(* IEC 61131-3 sources: PortalRobot/Portal_robot/Device/application/FB (part 4) *)

(* ---- FB_MAGAZINE.UpdateTypeStatus.st ---- *)
METHOD PRIVATE UpdateTypeStatus
VAR_IN_OUT
	stMagazineInventory : ST_MAGAZINE_INVENTORY;
END_VAR
VAR
	uiType : UINT; // Тип секции, 1..3
	uiSlot : UINT; // Проверяемый слот
	iSlot  : SINT; // Индекс массива содержимого
END_VAR

// --- BEGIN IMPLEMENTATION ---

FOR uiType := UINT#1 TO UINT#3 DO
	Status.stTypeStatus.aiBlankSlot[uiType] := SINT#0;
	Status.stTypeStatus.aiFreeSlot[uiType] := SINT#0;
	Status.stTypeStatus.auiBlankCount[uiType] := UINT#0;
	Status.stTypeStatus.auiDetailCount[uiType] := UINT#0;
	Status.stTypeStatus.auiFreeCount[uiType] := UINT#0;
END_FOR;

IF (iActiveSlotCount > SINT#0)
AND (uiTypeCount >= UINT#1)
AND (uiTypeCount <= UINT#3) THEN
	FOR uiSlot := UINT#1 TO SINT_TO_UINT(iActiveSlotCount) DO
		iSlot := UINT_TO_SINT(uiSlot);
		IF NOT stMagazineInventory.aSlots[iSlot].xInPosition THEN
			// Пустой слот универсален: тип 0
			// означает отсутствие изделия, а не запрет укладки конкретного типа.
			FOR uiType := UINT#1 TO uiTypeCount DO
				Status.stTypeStatus.auiFreeCount[uiType] :=
					Status.stTypeStatus.auiFreeCount[uiType] + UINT#1;
				IF Status.stTypeStatus.aiFreeSlot[uiType] = SINT#0 THEN
					Status.stTypeStatus.aiFreeSlot[uiType] := iSlot;
				END_IF;
			END_FOR;
		ELSE
			uiType := stMagazineInventory.aSlots[iSlot].uiProductType;
			IF (uiType >= UINT#1) AND (uiType <= uiTypeCount)
			AND (stMagazineInventory.aSlots[iSlot].eDetailType = E_DETAIL_TYPE.BLANK) THEN
				Status.stTypeStatus.auiBlankCount[uiType] :=
					Status.stTypeStatus.auiBlankCount[uiType] + UINT#1;
				IF Status.stTypeStatus.aiBlankSlot[uiType] = SINT#0 THEN
					Status.stTypeStatus.aiBlankSlot[uiType] := iSlot;
				END_IF;
			ELSIF (uiType >= UINT#1) AND (uiType <= uiTypeCount)
			AND (stMagazineInventory.aSlots[iSlot].eDetailType = E_DETAIL_TYPE.DETAIL) THEN
				Status.stTypeStatus.auiDetailCount[uiType] :=
					Status.stTypeStatus.auiDetailCount[uiType] + UINT#1;
			END_IF;
		END_IF;
	END_FOR;
END_IF;

(* ---- FB_MOTION_MANAGER.UpdateErrorView.st ---- *)
METHOD UpdateErrorView : ST_MOTION_MANAGER_ERROR
VAR_INPUT
	dwError : DWORD; // Битовая маска для расшифровки
END_VAR
VAR
	stError : ST_MOTION_MANAGER_ERROR; // Представление ошибок отдельными флагами
END_VAR

// --- BEGIN IMPLEMENTATION ---

stError.POINT_INVALID := (dwError AND ERR_POINT_INVALID) <> DWORD#0;
stError.GROUP_ERROR := (dwError AND ERR_GROUP) <> DWORD#0;
stError.GLOBAL_STOP := (dwError AND ERR_GLOBAL_STOP) <> DWORD#0;

UpdateErrorView := stError;

(* ---- FB_POINT_MANAGER.UpdateErrorView.st ---- *)
METHOD UpdateErrorView : ST_POINT_MANAGER_ERROR
VAR_INPUT
	dwError : DWORD; // Битовая маска для расшифровки
END_VAR
VAR
	stError : ST_POINT_MANAGER_ERROR; // Представление ошибок отдельными флагами
END_VAR

// --- BEGIN IMPLEMENTATION ---

stError.X_OUT_OF_LIMIT := (dwError AND X_OUT_OF_LIMIT) <> DWORD#0;
stError.Y_OUT_OF_LIMIT := (dwError AND Y_OUT_OF_LIMIT) <> DWORD#0;
stError.Z_OUT_OF_LIMIT := (dwError AND Z_OUT_OF_LIMIT) <> DWORD#0;
stError.INVALID_VEL := (dwError AND INVALID_VEL) <> DWORD#0;

UpdateErrorView := stError;

(* ---- FB_ROBOT.UpdateErrorView.st ---- *)
METHOD UpdateErrorView : ST_ROBOT_ERROR
VAR_INPUT
	dwError : DWORD; // Битовая маска для расшифровки
END_VAR
VAR
	stError : ST_ROBOT_ERROR; // Представление ошибок отдельными флагами
END_VAR

// --- BEGIN IMPLEMENTATION ---

stError.WRONG_ACTION := (dwError AND ERR_ROBOT_WRONG_ACTION) <> DWORD#0;
stError.MOTION_ERROR := (dwError AND ERR_ROBOT_MOTION) <> DWORD#0;
stError.GRIPPER_ERROR := (dwError AND ERR_ROBOT_GRIPPER) <> DWORD#0;
stError.MODBUS_ERROR := (dwError AND ERR_ROBOT_MODBUS_STUB) <> DWORD#0;
stError.STOP_ERROR := (dwError AND ERR_ROBOT_STOP) <> DWORD#0;

UpdateErrorView := stError;

(* ---- FB_TWO_PALLET.IsSignalConfigurationValid.st ---- *)
METHOD IsSignalConfigurationValid : BOOL
VAR_INPUT
	uiP1Signals : UINT;
	uiP2Signals : UINT;
END_VAR

// --- BEGIN IMPLEMENTATION ---

// Рабочее положение каждого цилиндра подтверждает ровно один геркон.
// Зацепление должно различать палеты и при опущенной П2 во время обмена.
IsSignalConfigurationValid := (uiP1Signals <= UINT#63)
	AND (uiP2Signals <= UINT#63)
	AND (((uiP1Signals AND UINT#3) = UINT#1) OR ((uiP1Signals AND UINT#3) = UINT#2))
	AND (((uiP2Signals AND UINT#3) = UINT#1) OR ((uiP2Signals AND UINT#3) = UINT#2))
	AND (((uiP1Signals AND UINT#12) = UINT#4) OR ((uiP1Signals AND UINT#12) = UINT#8))
	AND (((uiP2Signals AND UINT#12) = UINT#4) OR ((uiP2Signals AND UINT#12) = UINT#8))
	AND (((uiP1Signals AND UINT#48) = UINT#16) OR ((uiP1Signals AND UINT#48) = UINT#32))
	AND (((uiP2Signals AND UINT#48) = UINT#16) OR ((uiP2Signals AND UINT#48) = UINT#32))
	AND ((uiP1Signals AND UINT#60) <> (uiP2Signals AND UINT#60));

(* ---- FB_TWO_PALLET.UpdateErrorView.st ---- *)
METHOD UpdateErrorView : ST_TWO_PALLET_ERROR
VAR_INPUT
	dwError : DWORD;
END_VAR
VAR
	stError : ST_TWO_PALLET_ERROR;
END_VAR

// --- BEGIN IMPLEMENTATION ---

stError.DRIVE_ERROR := (dwError AND ERR_DRIVE) <> DWORD#0;
stError.SENSOR_CONTRADICTION := (dwError AND ERR_SENSOR_CONTRADICTION) <> DWORD#0;
stError.CYLINDER_TIMEOUT := (dwError AND ERR_CYLINDER_TIMEOUT) <> DWORD#0;
stError.MOTION_TIMEOUT := (dwError AND ERR_MOTION_TIMEOUT) <> DWORD#0;
stError.LOGIC_ERROR := (dwError AND ERR_LOGIC) <> DWORD#0;
stError.SEQUENCE_INTERRUPTED := (dwError AND ERR_SEQUENCE_INTERRUPTED) <> DWORD#0;

UpdateErrorView := stError;
